PROGRAM MB_SERVER_DEMO
VAR
	IP_CONTROL2_1: IP_CONTROL2;
	MB_SERVER_1: MB_SERVER;
	IP_C: IP_C;
	S_BUF: NETWORK_BUFFER_SHORT;
	R_BUF: NETWORK_BUFFER_SHORT;
	DATA: ARRAY [0..255] OF WORD;
	VMAP: ARRAY [1..10] OF VMAP_DATA;
END_VAR

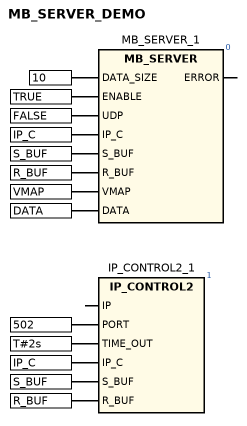
MB_SERVER_1(
    DATA_SIZE := 10,
    ENABLE := TRUE,
    UDP := FALSE,
    IP_C := IP_C,
    S_BUF := S_BUF,
    R_BUF := R_BUF,
    VMAP := VMAP,
    DATA := DATA); // MB_SERVER
IP_CONTROL2_1(PORT := 502, TIME_OUT := T#2s, IP_C := IP_C, S_BUF := S_BUF, R_BUF := R_BUF); // IP_CONTROL2

END_PROGRAM

(* stored: Version 1.1.0.1, ProductVersion 3.1.4024.9
   POU MB_SERVER_DEMO: Id {e3806b00-5f96-4dc3-a5c4-0e961f8b13c4}, SpecialFunc None *)
